Universal Robots PolyScope program: UR5e_Program.urp

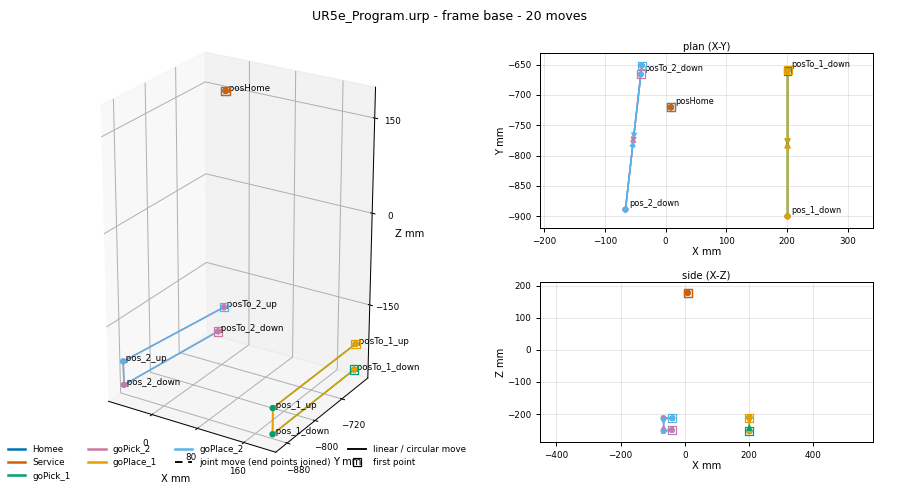
[picture p0: tool path of UR5e_Program.urp in frame base, 20 of 20 moves have a stored position in this frame; points joined in program order, loops and branches not executed]
Program OPCUA_LJ_Henrik_01.02.2023 (installation=OPC_UA_LJ_Henrik_Installation_01.02.2023 directory=/programs/usbdisk_0/WS2223_HSemdenleer_project/safe_03.02.2023 createdIn=5.8.0.10253 lastSavedIn=5.8.0.10253 robotSerialNumber=20205500995)
Calibrated DH parameters: a=[-0.000062, -0.131993, -0.388522, -0.000001, 0.000096, 0]; d=[0.162564, -380.047805, 374.673146, 5.508098, 0.099497, 0.099557]; alpha=[1.571156, -0.001063, 0.010019, 1.567513, -1.569344, 0]; deltaTheta=[0, 1.255078, 4.890399, 0.137715, -0.000001, -0.000001]
BeforeStart
  URCap Gripper Activate (Robotiq_Grippers, Robotiq Inc.) dataModel(ResetAndActivateKey=false)
  Base_var := Base_1
  Call Homee
  URCap OPC UA Server (OPC UA, Rocketfarm AS) dataModel(function=read, attributeName=start, attributeType=bool, selectedProgramVariable=start, Variable(key=newProgramVariable, variable(name=start)))
  URCap OPC UA Server (OPC UA, Rocketfarm AS) dataModel(function=read, onError=none, attributeName=isBusy, attributeType=bool, selectedProgramVariable=isBusy, Variable(key=newProgramVariable, variable(name=isBusy)))
  URCap OPC UA Server (OPC UA, Rocketfarm AS) dataModel(function=read, attributeName=service, attributeType=int, selectedProgramVariable=service, Variable(key=newProgramVariable, variable(name=service)))
  URCap OPC UA Server (OPC UA, Rocketfarm AS) dataModel(function=read, onError=none, attributeName=pick_id, attributeType=int, selectedProgramVariable=pick_id, Variable(key=newProgramVariable, variable(name=pick_id)))
  URCap OPC UA Server (OPC UA, Rocketfarm AS) dataModel(function=read, attributeName=pick_dir, attributeType=int, selectedProgramVariable=pick_dir, Variable(key=newProgramVariable, variable(name=pick_dir)))
  URCap OPC UA Server (OPC UA, Rocketfarm AS) dataModel(function=read, onError=none, attributeName=place_id, attributeType=int, selectedProgramVariable=place_id, Variable(key=newProgramVariable, variable(name=place_id)))
  URCap OPC UA Server (OPC UA, Rocketfarm AS) dataModel(function=read, attributeName=place_dir, attributeType=int, selectedProgramVariable=place_dir, Variable(key=newProgramVariable, variable(name=place_dir)))
Robot Program (runOnlyOnce=false)
  Call Homee
  Call openGripper
  Call Service
  Call wait_for_start
  Call read_pos
  Switch expression=pick_dir
    Case (caseValue=1)
      Base_var := Base_1
    Case (caseValue=2)
      Base_var := Base_2
    Case (caseValue=3)
      Halt
    Case (caseValue=4)
      Halt
    Case (caseValue=5)
      Halt
    Case (caseValue=6)
      Base_var := Base_6
    Case (caseValue=2147483647)
      Halt
  Call Homee
  Switch expression=pick_id
    Case (caseValue=1)
      Call goPick_1
    Case (caseValue=2)
      Call goPick_2
    Case (caseValue=101)
      'test'
    Case (caseValue=2147483647)
      Halt
  Call Homee
  Switch expression=place_dir
    Case (caseValue=1)
      Base_var := Base_1
    Case (caseValue=2)
      Base_var := Base_2
    Case (caseValue=3)
      Halt
    Case (caseValue=4)
      Halt
    Case (caseValue=5)
      Halt
    Case (caseValue=6)
      Base_var := Base_6
    Case (caseValue=2147483647)
      Halt
  Call Homee
  Switch expression=place_id
    Case (caseValue=1)
      Call goPlace_1
    Case (caseValue=2)
      Call goPlace_2
    Case (caseValue=101)
      'test'
    Case (caseValue=2147483647)
      Halt
SubProgram -> Service
SubProgram -> Homee
SubProgram -> openGripper
SubProgram -> wait_for_start
SubProgram -> read_pos
SubProgram -> goPick_1
SubProgram -> goPlace_1
SubProgram -> goPick_2
SubProgram -> goPlace_2
SubProgram Homee (keepSynchronizedWithDisk=false)
  MoveJ speed 60 deg/s, acceleration 40 deg/s^2 (useActiveTCP=false) tcp=Gipper_Plate; feature=Base_var
    Waypoint posHome: TCP in base x=9.035 y=-720.391 z=177.299 mm, rx=-0.0001 ry=-2.2215 rz=2.2215 rad; joints [-70.209, -113.29, -120.919, 234.12, -69.66, 180.484] deg; TCP offset x=0 y=-41.25 z=200.5 mm, rx=0 ry=0 rz=0 rad; feature pose in base x=579.871 y=-773.762 z=-332.712 mm, rx=-0.0008 ry=0.017 rz=-3.1361 rad
SubProgram openGripper (keepSynchronizedWithDisk=false)
  URCap Gripper (Robotiq_Grippers, Robotiq Inc.) dataModel(position=0.0, force=0.0, speed=20.0, positionInDouble=0.0, forceInDouble=0.0, speedInDouble=20.0, slaveIds=[9], blocking=true)
SubProgram Service (keepSynchronizedWithDisk=false)
  URCap OPC UA Server (OPC UA, Rocketfarm AS) dataModel(function=read, attributeName=service, attributeType=int, selectedProgramVariable=service, Variable(key=newProgramVariable, variable=service))
  Switch expression=service
    Case (caseValue=0)
      'no service needed'
    Case (caseValue=1)
      service := 0
      URCap OPC UA Server (OPC UA, Rocketfarm AS) dataModel(function=write, attributeName=service, attributeType=int, selectedProgramVariable=service, Variable(key=newProgramVariable, variable=service))
      Base_var := Base_1
      MoveJ speed 60 deg/s, acceleration 80 deg/s^2 (useActiveTCP=true) feature=Base_var
        Waypoint Waypoint_1: TCP in base x=9.085 y=-720.407 z=177.329 mm, rx=0 ry=2.2213 rz=-2.2214 rad; joints [-70.206, -113.289, -120.916, 234.119, -69.662, 180.485] deg; feature pose in base x=579.871 y=-773.762 z=-332.712 mm, rx=-0.0008 ry=0.017 rz=-3.1361 rad
      Halt
    Case (caseValue=2)
      service := 0
      URCap OPC UA Server (OPC UA, Rocketfarm AS) dataModel(function=write, attributeName=service, attributeType=int, selectedProgramVariable=service, Variable(key=newProgramVariable, variable=service))
      Base_var := Base_2
      MoveJ speed 60 deg/s, acceleration 80 deg/s^2 (useActiveTCP=true) feature=Base_var
        Waypoint Waypoint_1: TCP in base x=9.085 y=-720.407 z=177.329 mm, rx=0 ry=2.2213 rz=-2.2214 rad; joints [-70.206, -113.289, -120.916, 234.119, -69.662, 180.485] deg
      Halt
    Case (caseValue=3)
      service := 0
      URCap OPC UA Server (OPC UA, Rocketfarm AS) dataModel(function=write, attributeName=service, attributeType=int, selectedProgramVariable=service, Variable(key=newProgramVariable, variable=service))
      Halt
    Case (caseValue=4)
      service := 0
      URCap OPC UA Server (OPC UA, Rocketfarm AS) dataModel(function=write, attributeName=service, attributeType=int, selectedProgramVariable=service, Variable(key=newProgramVariable, variable=service))
      Halt
    Case (caseValue=5)
      service := 0
      URCap OPC UA Server (OPC UA, Rocketfarm AS) dataModel(function=write, attributeName=service, attributeType=int, selectedProgramVariable=service, Variable(key=newProgramVariable, variable=service))
      Halt
    Case (caseValue=6)
      service := 0
      URCap OPC UA Server (OPC UA, Rocketfarm AS) dataModel(function=write, attributeName=service, attributeType=int, selectedProgramVariable=service, Variable(key=newProgramVariable, variable=service))
      Base_var := Base_6
      MoveJ speed 60 deg/s, acceleration 80 deg/s^2 (useActiveTCP=true) feature=Base_var
        Waypoint Waypoint_1: TCP in base x=9.085 y=-720.407 z=177.329 mm, rx=0 ry=2.2213 rz=-2.2214 rad; joints [-70.206, -113.289, -120.916, 234.119, -69.662, 180.485] deg
      Halt
SubProgram wait_for_start (keepSynchronizedWithDisk=false)
  isBusy := False
  URCap OPC UA Server (OPC UA, Rocketfarm AS) dataModel(function=write, attributeName=isBusy, attributeType=bool, selectedProgramVariable=isBusy, Variable(key=newProgramVariable, variable=isBusy))
  URCap OPC UA Server (OPC UA, Rocketfarm AS) dataModel(function=read, onError=none, attributeName=start, attributeType=bool, selectedProgramVariable=start, Variable(key=newProgramVariable, variable(name=start)))
  Loop While (checkContinuously=false) expression=True ≠start
    Wait Sleep waitTime=0.1
    URCap OPC UA Server (OPC UA, Rocketfarm AS) dataModel(function=read, attributeName=start, attributeType=bool, selectedProgramVariable=start, Variable(key=newProgramVariable, variable=start))
  start := False
  URCap OPC UA Server (OPC UA, Rocketfarm AS) dataModel(function=write, attributeName=start, attributeType=bool, selectedProgramVariable=start, Variable(key=newProgramVariable, variable=start))
  isBusy := True
  URCap OPC UA Server (OPC UA, Rocketfarm AS) dataModel(function=write, attributeName=isBusy, attributeType=bool, selectedProgramVariable=isBusy, Variable(key=newProgramVariable, variable=isBusy))
SubProgram read_pos (keepSynchronizedWithDisk=false)
  pick_id := 0
  pick_dir := 0
  place_id := 0
  place_dir := 0
  URCap OPC UA Server (OPC UA, Rocketfarm AS) dataModel(function=read, onError=none, attributeName=pick_id, attributeType=int, selectedProgramVariable=pick_id, Variable(key=newProgramVariable, variable=pick_id))
  URCap OPC UA Server (OPC UA, Rocketfarm AS) dataModel(function=read, onError=none, attributeName=pick_dir, attributeType=int, selectedProgramVariable=pick_dir, Variable(key=newProgramVariable, variable=pick_dir))
  URCap OPC UA Server (OPC UA, Rocketfarm AS) dataModel(function=read, onError=none, attributeName=place_id, attributeType=int, selectedProgramVariable=place_id, Variable(key=newProgramVariable, variable=place_id))
  URCap OPC UA Server (OPC UA, Rocketfarm AS) dataModel(function=read, onError=none, attributeName=place_dir, attributeType=int, selectedProgramVariable=place_dir, Variable(key=newProgramVariable, variable=place_dir))
SubProgram goPick_1 (keepSynchronizedWithDisk=false)
  MoveP speed 250 mm/s, acceleration 1200 mm/s^2 (blendRadius=0.025 useActiveTCP=false) tcp=Gipper_Plate; feature=Base_var
    Waypoint posTo_1_down: TCP in base x=201.104 y=-660.658 z=-253.433 mm, rx=-0.005 ry=-2.2192 rz=2.2191 rad; joints [-41.966, -175.49, -99.442, 275.022, -41.087, 179.948] deg; feature pose in base x=579.871 y=-773.762 z=-332.712 mm, rx=-0.0008 ry=0.017 rz=-3.1361 rad
  MoveL speed 250 mm/s, acceleration 1200 mm/s^2 (useActiveTCP=false) tcp=Gipper_Plate; feature=Base_var
    Waypoint pos_1_down: TCP in base x=201.129 y=-900.06 z=-253.44 mm, rx=-0.0051 ry=-2.2193 rz=2.2191 rad; joints [-59.224, -182.264, -58.227, 240.365, -58.375, 180.373] deg
  URCap Gripper (Robotiq_Grippers, Robotiq Inc.) dataModel(position=45.0, force=0.0, speed=20.0, positionInDouble=45.0, forceInDouble=0.0, speedInDouble=20.0, slaveIds=[9], blocking=true)
  MoveL speed 250 mm/s, acceleration 1200 mm/s^2 (useActiveTCP=true) feature=Base_var
    Waypoint pos_1_up: TCP in base x=201.118 y=-900.058 z=-210.957 mm, rx=-0.005 ry=-2.2193 rz=2.2191 rad; joints [-59.221, -176.568, -63.853, 240.29, -58.371, 180.379] deg
  MoveL speed 250 mm/s, acceleration 1200 mm/s^2 (useActiveTCP=true) feature=Base_var
    Waypoint posTo_1_up: TCP in base x=201.144 y=-658.298 z=-210.983 mm, rx=-0.0049 ry=-2.2193 rz=2.2191 rad; joints [-41.696, -169.682, -104.754, 274.511, -40.821, 179.964] deg
SubProgram goPick_2 (keepSynchronizedWithDisk=false)
  MoveP speed 250 mm/s, acceleration 1200 mm/s^2 (blendRadius=0.025 useActiveTCP=true) feature=Base_var
    Waypoint posTo_2_down: TCP in base x=-40.775 y=-665.904 z=-249.643 mm, rx=-0.1214 ry=-2.1624 rz=2.1626 rad; joints [-69.935, -175.956, -106.192, 282.273, -62.841, 179.837] deg; feature pose in base x=579.871 y=-773.762 z=-332.712 mm, rx=-0.0008 ry=0.017 rz=-3.1361 rad
  MoveL speed 250 mm/s, acceleration 1200 mm/s^2 (useActiveTCP=true) feature=Base_var
    Waypoint pos_2_down: TCP in base x=-66.024 y=-888.588 z=-252.619 mm, rx=-0.1212 ry=-2.1624 rz=2.1626 rad; joints [-80.123, -179.285, -68.277, 247.569, -73.021, 180.208] deg
  URCap Gripper (Robotiq_Grippers, Robotiq Inc.) dataModel(position=45.0, force=0.0, speed=20.0, positionInDouble=45.0, forceInDouble=0.0, speedInDouble=20.0, slaveIds=[9], blocking=true)
  MoveL speed 250 mm/s, acceleration 1200 mm/s^2 (useActiveTCP=true) feature=Base_var
    Waypoint pos_2_up: TCP in base x=-66.05 y=-889.017 z=-213.025 mm, rx=-0.1214 ry=-2.1624 rz=2.1626 rad; joints [-80.125, -174.091, -73.051, 247.146, -73.019, 180.221] deg
  MoveL speed 250 mm/s, acceleration 1200 mm/s^2 (useActiveTCP=true) feature=Base_var
    Waypoint posTo_2_up: TCP in base x=-39.031 y=-651.457 z=-213.094 mm, rx=-0.1213 ry=-2.1624 rz=2.1626 rad; joints [-68.781, -171.364, -112.557, 284.053, -61.695, 179.818] deg
SubProgram goPlace_1 (keepSynchronizedWithDisk=false)
  MoveL speed 250 mm/s, acceleration 1200 mm/s^2 (useActiveTCP=true) feature=Base_var
    Waypoint posTo_1_up: TCP in base x=201.144 y=-658.298 z=-210.983 mm, rx=-0.0049 ry=-2.2193 rz=2.2191 rad; joints [-41.696, -169.682, -104.754, 274.511, -40.821, 179.964] deg; feature pose in base x=579.871 y=-773.762 z=-332.712 mm, rx=-0.0008 ry=0.017 rz=-3.1361 rad
  MoveL speed 250 mm/s, acceleration 1200 mm/s^2 (useActiveTCP=true) feature=Base_var
    Waypoint pos_1_up: TCP in base x=201.118 y=-900.058 z=-210.957 mm, rx=-0.005 ry=-2.2193 rz=2.2191 rad; joints [-59.221, -176.568, -63.853, 240.29, -58.371, 180.379] deg
  MoveL speed 250 mm/s, acceleration 1200 mm/s^2 (useActiveTCP=false) tcp=Gipper_Plate; feature=Base_var
    Waypoint pos_1_down: TCP in base x=201.129 y=-900.06 z=-253.44 mm, rx=-0.0051 ry=-2.2193 rz=2.2191 rad; joints [-59.224, -182.264, -58.227, 240.365, -58.375, 180.373] deg
  URCap Gripper (Robotiq_Grippers, Robotiq Inc.) dataModel(position=0.0, force=100.0, speed=100.0, positionInDouble=0.0, forceInDouble=100.0, speedInDouble=100.0, slaveIds=[9], blocking=true)
  MoveL speed 250 mm/s, acceleration 1200 mm/s^2 (useActiveTCP=true) feature=Base_var
    Waypoint posTo_1_down: TCP in base x=201.104 y=-660.658 z=-253.433 mm, rx=-0.005 ry=-2.2192 rz=2.2191 rad; joints [-41.966, -175.49, -99.442, 275.022, -41.087, 179.948] deg
SubProgram goPlace_2 (keepSynchronizedWithDisk=false)
  MoveP speed 250 mm/s, acceleration 1200 mm/s^2 (blendRadius=0.025 useActiveTCP=true) feature=Base_var
    Waypoint posTo_2_up: TCP in base x=-39.031 y=-651.457 z=-213.094 mm, rx=-0.1213 ry=-2.1624 rz=2.1626 rad; joints [-68.781, -171.364, -112.557, 284.053, -61.695, 179.818] deg; feature pose in base x=579.871 y=-773.762 z=-332.712 mm, rx=-0.0008 ry=0.017 rz=-3.1361 rad
  MoveL speed 250 mm/s, acceleration 1200 mm/s^2 (useActiveTCP=true) feature=Base_var
    Waypoint pos_2_up: TCP in base x=-66.05 y=-889.017 z=-213.025 mm, rx=-0.1214 ry=-2.1624 rz=2.1626 rad; joints [-80.125, -174.091, -73.051, 247.146, -73.019, 180.221] deg
  MoveL speed 250 mm/s, acceleration 1200 mm/s^2 (useActiveTCP=true) feature=Base_var
    Waypoint pos_2_down: TCP in base x=-66.024 y=-888.588 z=-252.619 mm, rx=-0.1212 ry=-2.1624 rz=2.1626 rad; joints [-80.123, -179.285, -68.277, 247.569, -73.021, 180.208] deg
  URCap Gripper (Robotiq_Grippers, Robotiq Inc.) dataModel(position=0.0, force=0.0, speed=20.0, positionInDouble=0.0, forceInDouble=0.0, speedInDouble=20.0, slaveIds=[9], blocking=true)
  MoveP speed 250 mm/s, acceleration 1200 mm/s^2 (blendRadius=0.025 useActiveTCP=true) feature=Base_var
    Waypoint posTo_2_down: TCP in base x=-40.775 y=-665.904 z=-249.643 mm, rx=-0.1214 ry=-2.1624 rz=2.1626 rad; joints [-69.935, -175.956, -106.192, 282.273, -62.841, 179.837] deg
